FUNCTION_BLOCK TrapezoIDal_velocity_trajectory
VAR_INPUT
	t0,q0,q1:lreal;
	a_max,v_max:lreal;
	t:lreal;
END_VAR
VAR_OUTPUT
	pos:lreal;
	vel:lreal;
	acc:lreal;
	finished:BOOL;
END_VAR
VAR
	h,V_v,A_a:lreal;
	Tp,Ta:lreal;
	t1:lreal;
END_VAR


h:=q1-q0;

V_v:=V_max;
A_a:=A_max;
IF(h<0) THEN
    V_v:=-V_max;
    A_a:=-A_max;
END_IF


//%step1,根据给定参数，计算加速时间、总时间
IF(ABS(h)>=(V_v*V_v/ABS(A_a))) THEN
    Tp:=(h*A_a+V_v*V_v)/(A_a*V_v);
    Ta:=V_v/A_a; 
	t1:=t0+Tp;
	
	IF (t>t0) AND (t<=t0+Ta) THEN
		pos:=q0+0.5*A_a*EXPT(t-t0,2);
        vel:=A_a*(t-t0);
        acc:=A_a;	
	ELSIF (t>t0+Ta) AND (t<=t1-Ta) THEN
		pos:=q0+A_a*Ta*(t-t0-Ta/2);
        vel:=A_a*Ta;
        acc:=0;	
	ELSIF (t<=t1) THEN
		pos:=q1-0.5*A_a*EXPT(t1-t,2);
        vel:=A_a*(t1-t);
        acc:=-A_a;	
	END_IF
   
	IF (t>t1) THEN
		finished:=TRUE;
		pos:=q1;
		vel:=0;
		acc:=0;
	ELSE
		finished:=FALSE;
	END_IF
	
	
ELSE	
    //%step2,没有匀速阶段
    Ta:=SQRT(h/A_a);
    Tp:=2*Ta;
	t1:=t0+Tp;
	
	IF (t>t0) AND (t<=(t0+Ta)) THEN
		pos:=q0+0.5*A_a*EXPT((t-t0),2);
        vel:=A_a*(t-t0);
        acc:=A_a;
	ELSIF (t<=t1) THEN
		pos:=q1-0.5*A_a*EXPT(t1-t,2);
        vel:=A_a*(t1-t);
        acc:=-A_a;
	END_IF
		
	IF (t>t1) THEN
		finished:=TRUE;
		pos:=q1;
		vel:=0;
		acc:=0;
	ELSE
		finished:=FALSE;
	END_IF
		
END_IF

END_FUNCTION_BLOCK

(* stored: Version 1.1.0.1, ProductVersion 3.1.4024.12
   POU TrapezoIDal_velocity_trajectory: Id {40b394c2-ad7f-4060-aa1b-5902f6e4807c}, SpecialFunc None *)
